Staubli VAL3: buildList.pgx

program buildList()
  local num i
  local string l_sPalletName
  local num l_nPosition[4]
  local string l_sEmpty
  local num l_nSize
begin
  // INIT the list
  l_sEmpty=""
  call use:stringCopy(l_sEmpty,sList)
  //
  // Build the list
  //
  for i=0 to size(sPalletName)-1
    // scan all
    if sPalletName[i]!=""
      l_sPalletName=sPalletName[i]
      call pallet:getPalletPos(l_sPalletName,l_nPosition)
      call pallet:getSizePallet(l_sPalletName,l_nSize)
      call use:strfill(l_sPalletName,12,l_sPalletName)
      call listAdd(l_sPalletName+"> "+toString("",l_nPosition+1)+"/"+toString("",l_nSize))
    endIf
  endFor
  // refresh it
  // rebuild the list
  call use:listempty()
  call use:listadd(sList)
end
